FUNCTION_BLOCK F_FRACTION_TO_PERCENT (* Anteil (REAL 0.0-1.0, von F_PWM_RAW_TO_PERCENT.OUT) in Prozent (REAL 0.0-100.0, fuer OPC-UA-Publish) umrechnen *)
  (* Standard: 61499-2; Description: Copyright (c) 2026 Meisterschulen am Ostbahnhof This program and the accompanying materials are made available under the terms of the Eclipse Public License 2.0 which is available at https://www.eclipse.org/legal/epl-2.0/ SPDX-License-Identifier: EPL-2.0 *)
  (* Version 1.0, 2026-08-28, Franz Höpfinger, Meisterschulen am Ostbahnhof, initial API and implementation and/or initial documentation *)
  PACKAGE logiBUS::signalprocessing::fieldbus;
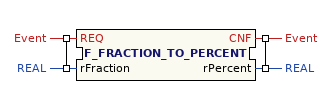
  EVENT_INPUT
    REQ WITH rFraction; (* Umrechnung anfordern *)
  END_EVENT
  EVENT_OUTPUT
    CNF WITH rPercent; (* Umrechnung abgeschlossen *)
  END_EVENT
  VAR_INPUT
    rFraction : REAL; (* Anteil 0.0-1.0 *)
  END_VAR
  VAR_OUTPUT
    rPercent : REAL; (* Prozentwert 0.0-100.0 *)
  END_VAR
  EC_STATES
    REQ : REQ -> CNF;
  END_STATES
  ALGORITHM REQ IN ST: (* 1.0 entspricht 100.0 % *)
rPercent := rFraction * 100.0;
  END_ALGORITHM
END_FUNCTION_BLOCK
